// TIA Portal V19 export
DATA_BLOCK "Data"   // DB40
// stored: Access Published, MemoryReserve 100, Namespace Global
   VAR
      general : "LAF_typeGeneralStatus";   // Global status information
      unit : "LAF_typeUnitInterface";   // Global information of units
   END_VAR
BEGIN
   // general.enablePower : Global power is off / Global Power ist ausgeschaltet
END_DATA_BLOCK
